// TIA Portal V19 export
DATA_BLOCK "Generic"   // DB60
// stored: Access Published, InstanceOfName Generic_FB, InstanceOfType FB
"Generic_FB"
   // VAR_INPUT
   //    AreaInterface1 : "AreaInterface";
   //    AreaInterface2 : "AreaInterface";
   //    AreaInterface3 : "AreaInterface";
   //    AreaInterface4 : "AreaInterface";
   // END_VAR
   // VAR_OUTPUT
   //    MachineInterface1 : "MachineInterface";
   //    MachineInterface2 : "MachineInterface";
   //    MachineInterface3 : "MachineInterface";
   //    MachineInterface4 : "MachineInterface";
   // END_VAR
   // VAR
   //    Ctrl : Struct
   //       RstAlarms : Bool;
   //    END_STRUCT;
   //    Sts : Struct
   //       Standstill : Bool;
   //       AlarmsPresence_GEN : Bool;
   //       AlarmsPresence_A01_2 : Bool;
   //       AlarmsPresence_A03_4 : Bool;
   //       WarningsPresence : Bool;
   //    END_STRUCT;
   //    Alarm : Struct
   //       CC1_PorteAperte : Bool;
   //       CC1_ThermalTrip_24Vdc_PLC_SINAMICS : Bool;
   //       CC1_ThermalTrip_24Vdc_Valves : Bool;
   //       CC1_ProtezioneElettronicaSitop : Bool;
   //       CC1_LowAirPressure : Bool;
   //       Area01_Aspo_LowAirPressure : Bool;
   //       Area02_03_Accopiamento_LowAirPressure : Bool;
   //       Area03_Pareggiamneto_LowAirPressure : Bool;
   //       Area04_Navetta_LowAirPressure : Bool;
   //       INFEED_640A1 : "InfeedAlr";
   //       CU_580A1 : "SinamicsCU_Alarms";
   //       CU_585A1 : "SinamicsCU_Alarms";
   //       CU_590A1 : "SinamicsCU_Alarms";
   //       CU_595A1 : "SinamicsCU_Alarms";
   //       CU_600A1 : "SinamicsCU_Alarms";
   //       CU_605A1 : "SinamicsCU_Alarms";
   //       CU_610A1 : "SinamicsCU_Alarms";
   //       CU_615A1 : "SinamicsCU_Alarms";
   //       PNDiag_ET200S_460A1 : "PnDiag_Alr";
   //       PNDiag_ET200S_490A1 : "PnDiag_Alr";
   //       PNDiag_ET200S_510A1 : "PnDiag_Alr";
   //       PNDiag_ET200S_530A1 : "PnDiag_Alr";
   //       PNDiag_ET200S_550A1 : "PnDiag_Alr";
   //       PNDiag_CU_580A1 : "PnDiag_Alr";
   //       PNDiag_CU_585A1 : "PnDiag_Alr";
   //       PNDiag_CU_590A1 : "PnDiag_Alr";
   //       PNDiag_CU_595A1 : "PnDiag_Alr";
   //       PNDiag_CU_600A1 : "PnDiag_Alr";
   //       PNDiag_CU_605A1 : "PnDiag_Alr";
   //       PNDiag_CU_610A1 : "PnDiag_Alr";
   //       PNDiag_CU_615A1 : "PnDiag_Alr";
   //       PnDiag_ENC_694P1 { S7_SetPoint := 'True'} : "PnDiag_Alr";
   //       PnDiag_ENC_894P1 { S7_SetPoint := 'True'} : "PnDiag_Alr";
   //       PnDiag_ENC_984P1 { S7_SetPoint := 'True'} : "PnDiag_Alr";
   //       PnDiag_ENC_994P1 { S7_SetPoint := 'True'} : "PnDiag_Alr";
   //       PnDiag_ENC_1004P1 { S7_SetPoint := 'True'} : "PnDiag_Alr";
   //       PnDiag_ENC_1008P1 { S7_SetPoint := 'True'} : "PnDiag_Alr";
   //       PnDiag_ENC_1034P1 { S7_SetPoint := 'True'} : "PnDiag_Alr";
   //       PnDiag_ENC_1044P1 { S7_SetPoint := 'True'} : "PnDiag_Alr";
   //       PnDiag_ENC_1074P1 { S7_SetPoint := 'True'} : "PnDiag_Alr";
   //       PnDiag_ENC_1088P1 { S7_SetPoint := 'True'} : "PnDiag_Alr";
   //       PnDiag_ENC_1093P1 { S7_SetPoint := 'True'} : "PnDiag_Alr";
   //       PnDiag_ENC_1124P1 { S7_SetPoint := 'True'} : "PnDiag_Alr";
   //       PnDiag_ENC_1138P1 { S7_SetPoint := 'True'} : "PnDiag_Alr";
   //       PnDiag_ENC_1143P1 { S7_SetPoint := 'True'} : "PnDiag_Alr";
   //       PnDiag_ENC_1844P1 { S7_SetPoint := 'True'} : "PnDiag_Alr";
   //       PnDiag_ENC_1853P1 { S7_SetPoint := 'True'} : "PnDiag_Alr";
   //       PnDiag_ENC_1858P1 { S7_SetPoint := 'True'} : "PnDiag_Alr";
   //       PnDiag_ENC_1863P1 { S7_SetPoint := 'True'} : "PnDiag_Alr";
   //       PnDiag_ENC_1868P1 { S7_SetPoint := 'True'} : "PnDiag_Alr";
   //       PnDiag_ENC_1903P1 { S7_SetPoint := 'True'} : "PnDiag_Alr";
   //       PnDiag_ENC_1908P1 { S7_SetPoint := 'True'} : "PnDiag_Alr";
   //       PnDiag_ENC_1913P1 { S7_SetPoint := 'True'} : "PnDiag_Alr";
   //       PnDiag_ENC_1918P1 { S7_SetPoint := 'True'} : "PnDiag_Alr";
   //       PnDiag_ENC_2264P1 { S7_SetPoint := 'True'} : "PnDiag_Alr";
   //       PnDiag_ENC_2284P1 { S7_SetPoint := 'True'} : "PnDiag_Alr";
   //       PnDiag_ENC_2374P1 { S7_SetPoint := 'True'} : "PnDiag_Alr";
   //       PnDiag_ENC_2394P1 { S7_SetPoint := 'True'} : "PnDiag_Alr";
   //       PnDiag_ENC_2404P1 { S7_SetPoint := 'True'} : "PnDiag_Alr";
   //       PnDiag_ENC_2434P1 { S7_SetPoint := 'True'} : "PnDiag_Alr";
   //       PnDiag_ENC_2464P1 { S7_SetPoint := 'True'} : "PnDiag_Alr";
   //       PnDiag_ENC_2534P1 { S7_SetPoint := 'True'} : "PnDiag_Alr";
   //       PnDiag_PAC_100A1 { S7_SetPoint := 'True'} : "PnDiag_Alr";
   //    END_STRUCT;
   //    Warning : Struct
   //       NoAutReady : Bool;
   //       CC1_ThermalTrip220V_ServiceSockets : Bool;
   //       CC1_ThermalTrip_Cooling1 : Bool;
   //       CC1_ThermalTrip_Cooling2 : Bool;
   //       JB001_ThermalTrip_Cooling : Bool;
   //       CC1_MaxTemperature : Bool;
   //       JB001_MaxTemperature : Bool;
   //       CC1_GuastoCondizionatore_1 : Bool;
   //       CC1_GuastoCondizionatore_2 : Bool;
   //       SitopUp_BatteriaScarica : Bool;
   //       SitopUp_BatteriaNonCarica : Bool;
   //       SitopUp_AllarmeBatteria : Bool;
   //       ScalanceXC116_1_NotOk : Bool;
   //       ScalanceXC116_2_NotOk : Bool;
   //       ScalanceXC216_NotOk : Bool;
   //       ScalanceSC632_NotOk : Bool;
   //       INFEED_640A1 : "InfeedWng";
   //       CU_580A1 : "SinamicsCU_Warnings";
   //       CU_585A1 : "SinamicsCU_Warnings";
   //       CU_590A1 : "SinamicsCU_Warnings";
   //       CU_595A1 : "SinamicsCU_Warnings";
   //       CU_600A1 : "SinamicsCU_Warnings";
   //       CU_605A1 : "SinamicsCU_Warnings";
   //       CU_610A1 : "SinamicsCU_Warnings";
   //       CU_615A1 : "SinamicsCU_Warnings";
   //    END_STRUCT;
   //    Diag : Struct
   //       CC1_INFEED_460A1 : "TO_Diagnostic";
   //       CU_580A1 { S7_SetPoint := 'True'} : "TO_Diagnostic";
   //       CU_585A1 { S7_SetPoint := 'True'} : "TO_Diagnostic";
   //       CU_590A1 { S7_SetPoint := 'True'} : "TO_Diagnostic";
   //       CU_595A1 { S7_SetPoint := 'True'} : "TO_Diagnostic";
   //       CU_600A1 { S7_SetPoint := 'True'} : "TO_Diagnostic";
   //       CU_605A1 { S7_SetPoint := 'True'} : "TO_Diagnostic";
   //       CU_610A1 { S7_SetPoint := 'True'} : "TO_Diagnostic";
   //       CU_615A1 { S7_SetPoint := 'True'} : "TO_Diagnostic";
   //    END_STRUCT;
   //    INFEED_640A1 : "Infeed";
   //    CU_580A1 : "SinamicsCU_Modulblock";
   //    CU_585A1 : "SinamicsCU_Modulblock";
   //    CU_590A1 : "SinamicsCU_Modulblock";
   //    CU_595A1 : "SinamicsCU_Modulblock";
   //    CU_600A1 : "SinamicsCU_Modulblock";
   //    CU_605A1 : "SinamicsCU_Modulblock";
   //    CU_610A1 : "SinamicsCU_Modulblock";
   //    CU_615A1 : "SinamicsCU_Modulblock";
   //    PnDiag_ET200S_460A1 : "PnDiag";
   //    PnDiag_ET200S_490A1 : "PnDiag";
   //    PnDiag_ET200S_510A1 : "PnDiag";
   //    PnDiag_ET200S_530A1 : "PnDiag";
   //    PnDiag_ET200S_550A1 : "PnDiag";
   //    PnDiag_CU_580A1 : "PnDiag";
   //    PnDiag_CU_585A1 : "PnDiag";
   //    PnDiag_CU_590A1 : "PnDiag";
   //    PnDiag_CU_595A1 : "PnDiag";
   //    PnDiag_CU_600A1 : "PnDiag";
   //    PnDiag_CU_605A1 : "PnDiag";
   //    PnDiag_CU_610A1 : "PnDiag";
   //    PnDiag_CU_615A1 : "PnDiag";
   //    PnDiag_ENC_694P1 { S7_SetPoint := 'True'} : "PnDiag";
   //    PnDiag_ENC_894P1 { S7_SetPoint := 'True'} : "PnDiag";
   //    PnDiag_ENC_984P1 { S7_SetPoint := 'True'} : "PnDiag";
   //    PnDiag_ENC_994P1 { S7_SetPoint := 'True'} : "PnDiag";
   //    PnDiag_ENC_1004P1 { S7_SetPoint := 'True'} : "PnDiag";
   //    PnDiag_ENC_1008P1 { S7_SetPoint := 'True'} : "PnDiag";
   //    PnDiag_ENC_1034P1 { S7_SetPoint := 'True'} : "PnDiag";
   //    PnDiag_ENC_1044P1 { S7_SetPoint := 'True'} : "PnDiag";
   //    PnDiag_ENC_1074P1 { S7_SetPoint := 'True'} : "PnDiag";
   //    PnDiag_ENC_1088P1 { S7_SetPoint := 'True'} : "PnDiag";
   //    PnDiag_ENC_1093P1 { S7_SetPoint := 'True'} : "PnDiag";
   //    PnDiag_ENC_1124P1 { S7_SetPoint := 'True'} : "PnDiag";
   //    PnDiag_ENC_1138P1 { S7_SetPoint := 'True'} : "PnDiag";
   //    PnDiag_ENC_1143P1 { S7_SetPoint := 'True'} : "PnDiag";
   //    PnDiag_ENC_1844P1 { S7_SetPoint := 'True'} : "PnDiag";
   //    PnDiag_ENC_1853P1 { S7_SetPoint := 'True'} : "PnDiag";
   //    PnDiag_ENC_1858P1 { S7_SetPoint := 'True'} : "PnDiag";
   //    PnDiag_ENC_1863P1 { S7_SetPoint := 'True'} : "PnDiag";
   //    PnDiag_ENC_1868P1 { S7_SetPoint := 'True'} : "PnDiag";
   //    PnDiag_ENC_1903P1 { S7_SetPoint := 'True'} : "PnDiag";
   //    PnDiag_ENC_1908P1 { S7_SetPoint := 'True'} : "PnDiag";
   //    PnDiag_ENC_1913P1 { S7_SetPoint := 'True'} : "PnDiag";
   //    PnDiag_ENC_1918P1 { S7_SetPoint := 'True'} : "PnDiag";
   //    PnDiag_ENC_2264P1 { S7_SetPoint := 'True'} : "PnDiag";
   //    PnDiag_ENC_2284P1 { S7_SetPoint := 'True'} : "PnDiag";
   //    PnDiag_ENC_2374P1 { S7_SetPoint := 'True'} : "PnDiag";
   //    PnDiag_ENC_2394P1 { S7_SetPoint := 'True'} : "PnDiag";
   //    PnDiag_ENC_2404P1 { S7_SetPoint := 'True'} : "PnDiag";
   //    PnDiag_ENC_2434P1 { S7_SetPoint := 'True'} : "PnDiag";
   //    PnDiag_ENC_2464P1 { S7_SetPoint := 'True'} : "PnDiag";
   //    PnDiag_ENC_2534P1 { S7_SetPoint := 'True'} : "PnDiag";
   //    PnDiag_PAC_100A1 { S7_SetPoint := 'True'} : "PnDiag";
   //    TON_CheckHighTemperatureCC1 : IEC_TIMER;
   //    TON_CheckHighTemperatureJB001 : IEC_TIMER;
   //    TOF_TurnOffConditionerCC1 : IEC_TIMER;
   //    TOF_TurnOffConditionerJB001 : IEC_TIMER;
   //    TON_Area02_03_Accoppiamento_Pressione_Aria_OK { S7_SetPoint := 'True'} : IEC_TIMER;
   //    TON_Area03_Pareggiamneto_Pressione_Aria_OK { S7_SetPoint := 'True'} : IEC_TIMER;
   //    TON_Area04_Navetta_Pressione_Aria_OK { S7_SetPoint := 'True'} : IEC_TIMER;
   // END_VAR
BEGIN
END_DATA_BLOCK
